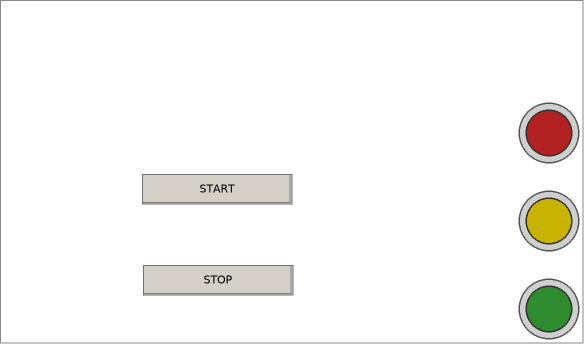
VISUALIZATION Visualization  // 584x344
    Lamp1 (514,98 70x70), variable: GVL.Red, style: Lamp-Lamp1-Red
    Lamp1 (514,186 70x70), variable: GVL.Yellow, style: Lamp-Lamp1-Yellow
    Lamp1 (514,274 70x70), variable: GVL.Green, style: Lamp-Lamp1-Green
    Button (142,174 150x30), "START"
        tap GVL.bStart
    Button (143,265 150x30), "STOP"
        tap GVL.bStop
END_VISUALIZATION

(* stored: Version 1.1.0.1, ProductVersion 3.1.4024.12
   Visu Visualization: Id {45de9aca-c94b-40e7-b30c-25001291a9af} *)
